PROGRAM P_Template_SAFETY
VAR_INPUT
	eMachineMode							: E_MachineMode; 		// Machine mode
	eMachineCommand							: E_MachineCommand; 	// Command from top level state program
END_VAR
VAR_OUTPUT
	eMachineState							: E_MachineState;
  	bError									: BOOL;
END_VAR
VAR
	// INPUTS
	bResetBusy								: BOOL;
	// OUTPUTS
	bResetCMD								: BOOL;
	// FBs
	rtRestart								: R_TRIG;
	rtReset									: R_TRIG;
	ftFinish								: F_TRIG;
	bSTOStatus								: BOOL;
	bSOSStatus								: BOOL;
	bAllAxisInSafeState						: BOOL;
	bAllAxisReady							: BOOL;
END_VAR

// =================== Inputs ===================
// Read input signals
Act_InUpdate();

// Error collection
Act_Error();
// ==============================================
rtReset(CLK:= eMachineCommand = E_MachineCommand.eReset, Q=> );
rtRestart(CLK:= eMachineCommand = E_MachineCommand.eRestart, Q=> );
ftFinish(CLK:= bResetBusy, Q=> );

IF bError THEN
	eMachineState								:= E_MachineState.eError;
END_IF

IF rtRestart.Q THEN
	eMachineState								:= E_MachineState.eRestarting;
	bResetCMD									:= TRUE;
END_IF

IF rtReset.Q THEN
	eMachineState								:= E_MachineState.eReseting;
	bResetCMD									:= TRUE;
END_IF

IF ftFinish.Q THEN
	eMachineState								:= E_MachineState.eRunning;
	bResetCMD									:= FALSE;
END_IF

// =================== Outputs ==================
Act_OutUpdate();
// ==============================================

ACTION Act_Error:
// Program summary error
bError 							:= 	(GVL_IO.dwAXErrors OR GVL_IO.dwGroupErrors) <> 0;
// OR bError 							:= GVL_IO.bSAFETY_Error;
END_ACTION

ACTION Act_InUpdate:
bResetBusy 						:= GVL_IO.bSAFETY_ResetBusy;
bSTOStatus  					:= GVL_IO.dwAXStatesSTO = 2#11_1111;
bSOSStatus  					:= GVL_IO.dwAXStatesSOS = 2#1111;
bAllAxisInSafeState  			:= (GVL_IO.dwAXStatesSTO OR GVL_IO.dwAXStatesSOS) = 2#11_1111;
bAllAxisReady 					:= (GVL_IO.dwAXStatesSTO OR GVL_IO.dwAXStatesSOS) = 0;
END_ACTION

ACTION Act_OutUpdate:
GVL_IO.bSAFETY_ResetCMD 		:= bResetCMD;
END_ACTION

END_PROGRAM

(* stored: Version 1.1.0.1, ProductVersion 3.1.4022.12
   POU P_Template_SAFETY: Id {1cf2eb24-e212-4be6-85ed-5951ec0bf36a}, SpecialFunc None
   Action Act_Error: Id {e5ac91da-f19a-412d-8637-7ec6e55e64b6}
   Action Act_InUpdate: Id {0b86017d-eb0b-4d2e-98d9-a259f7a022eb}
   Action Act_OutUpdate: Id {d32cba82-d123-4275-bbd9-98ad77c0c152} *)
